// TIA Portal V21 export
VAR_GLOBAL   // PLC tag table "KAllMotore"
END_VAR
VAR_GLOBAL CONSTANT   // user constants
   KAllMot_EncMismatch : Int := 1;
   KAllMot_ToutMovimento : Int := 2;
   KAllMot_InverterFault : Int := 3;
   KAllMot_TermicoVentola : Int := 4;
   KAllMot_RotturaCinghia : Int := 5;
   KAllMot_TimeOutAnticaduta : Int := 6;
   KAllMot_Freno : Int := 7;
   KAllMot_Freno2 : Int := 8;
   KAllMot_ComunInverter : Int := 9;
   KAllMot_ComunEncoder : Int := 10;
   KAllMot_TOutMarcia : Int := 11;
   KAllMot_ConteggioEnc : Int := 12;
   KAllMot_FolError : Int := 13;
   KAllMot_Bloccato : Int := 14;
   KAllMot_TroppoVeloce : Int := 15;
   KAllMot_SpinaSicNoInPos : Int := 32;
   "KAllMot_22(Word1_x6)" : Int := 22;
   "KAllMot_23(Word1_x7)" : Int := 23;
END_VAR
